FUNCTION_BLOCK aFb_Motor
VAR_INPUT
	Mode: aE_Mode := aE_Mode.Auto;
	
	//Manual
	Start: BOOL;
	Stop: BOOL;
	SetSpeed: REAL;
	Reset1: BOOL;
	
	//Auto
	RunCondition: BOOL;
	StopCondition: BOOL;
	SpeedCondition: REAL;
	
	//Others
	RunFeedback: BOOL;
	Interlock: BOOL;
	Maxspeed: REAL:= 1500;
	ActualSpeed: REAL;
END_VAR
VAR_OUTPUT
	Cmd: BOOL;
	Fault: BOOL;
	State: aE_State;
	Speed: REAL;
	Runtime: UDINT := 0;
	AccRuntime: UDINT := 0;
END_VAR
VAR
	{attribute 'hide'}
	fbTon: TON;
	{attribute 'hide'}
	fbTRuntime: TON;
END_VAR

CASE Mode OF 
	aE_Mode.Manual: 
		Cmd := (Cmd OR Start) AND NOT Stop AND NOT Fault AND NOT Interlock;
		IF Cmd THEN
			State := aE_State.ManRun;
		ELSE
			State := aE_State.ManStop;
		END_IF
	aE_Mode.Auto:
		Cmd := (Cmd OR RunCondition) AND NOT StopCondition AND NOT Fault AND NOT Interlock;
		State := aE_State.Auto;
	aE_Mode.Service:
		Cmd := (Cmd OR Start) AND NOT Stop AND NOT Fault;
END_CASE

IF Cmd THEN
	IF Mode = aE_Mode.Auto THEN
		Speed := LIMIT(-Maxspeed, SpeedCondition, Maxspeed);
	ELSE
		Speed := LIMIT(-Maxspeed, SetSpeed, Maxspeed);
	END_IF
ELSE 
	Speed:= 0;
END_IF

fbTon(IN := Cmd, PT := T#5S);
IF fbTon.Q AND NOT RunFeedback THEN
	Fault := TRUE;
	State := aE_State.Fault;
END_IF

IF Reset1 THEN
	Fault := FALSE;
END_IF

IF Cmd THEN
	fbTRuntime(IN := NOT fbTRuntime.Q, PT:= T#1S);
	IF fbTRuntime.Q THEN
		Runtime:= Runtime + 1;
		AccRuntime := AccRuntime + 1;
	END_IF
ELSE
	Runtime:= 0;
END_IF

END_FUNCTION_BLOCK

(* stored: Version 1.1.0.1, ProductVersion 3.1.4024.4
   POU aFb_Motor: Id {deea6eae-00c4-4d52-adc2-0d6a9e27c1a4}, SpecialFunc None *)
